Staubli VAL3: moveTo.pgx

public program moveTo(tool x_tTool, mdesc x_mDesc, num x_nMoveType, bool& x_bUnreached[], joint& x_jJoint[], num& x_nMoveId)
begin
  //
  // use the percentage speed
  //
  x_mDesc.vel=saveData:nSpeed/100*x_mDesc.vel
  x_nMoveId=movej(x_jJoint,x_tTool,x_mDesc)
end
